PROGRAM PRG_IP1_ECAT_Interfaces
VAR
END_VAR

ROUGH1_VRC_01_AtOpnLS := TMO_ROUGH1_VRC_01.iq_stValve.i_xOpnLS;
ROUGH2_VRC_01_AtOpnLS := TMO_ROUGH2_VRC_01.iq_stValve.i_xOpnLS;

END_PROGRAM

(* stored: Version 1.1.0.1, ProductVersion 3.1.4022.18
   POU PRG_IP1_ECAT_Interfaces: Id {e21a7b5a-d65b-44a4-910d-0603adcdae6b}, SpecialFunc None *)
